// TIA Portal V20 export
// export: Created 2025-12-01T14:57:41.0235932Z, ExportSetting None, DisplayName Totally Integrated Automation Portal, DisplayVersion V20 Update 3, DisplayName TIA Portal Openness, DisplayVersion V20 Update 3, DisplayName TIA Portal Version Control Interface, DisplayVersion V20 Update 3, DisplayName STEP 7 Professional, DisplayVersion V20 Update 3, DisplayName STEP 7 Safety, DisplayVersion V20 Update 2, DisplayName WinCC Basic/Comfort/Advanced, DisplayVersion V20 Update 3, DisplayName WinCC Professional, DisplayVersion V20 Update 3, DisplayName WinCC Unified, DisplayVersion V20 Update 3
FUNCTION_BLOCK "FB385_Operaciones_Paletizador_NDD"   // FB385, LAD
{ S7_Optimized_Access := 'FALSE' }
// stored: AutoNumber false, SetENOAutomatically false
   VAR_INPUT
      MesaElevador : UInt;
      MesaGarra : UInt;
      MesaHorquilla : UInt;
      ZonaCajon_Libre : Bool;
      ElevadorEnReposo : Bool;
      ElevadorPaletizando : Bool;
      DesHabilitar_Horquilla : Bool;
      DesHabilitar_Garra : Bool;
   END_VAR
   VAR_IN_OUT
      Horquilla : "NDD_Interlock_Horquilla";
      Garra : "NDD_Interlock_Garras";
      TELEV : "NDD_Interlock_TElev";
      Ordenes : "NDD_Ordenes";
   END_VAR
   VAR
      ControlUT_MesaElevador : "UDT_UTs_Control";
      DatosUT_MesaElevador { S7_SetPoint := 'True'} : "UDT_UTs_Datos";
      ControlUT_MesaGarra { S7_SetPoint := 'True'} : "UDT_UTs_Control";
      ControlUT_MesaHorquilla { S7_SetPoint := 'True'} : "UDT_UTs_Control";
      UT_MesaElevador : UInt;
      UT_MesaGarra : UInt;
      UT_MesaHorquilla : UInt;
      DesHabilitar_NDD : Bool;
      ExisteUT_MTElev { ExternalAccessible := 'False'; ExternalVisible := 'False'; ExternalWritable := 'False'} : Bool;
      TElev_PaletizarPaleta : Bool;
      TElev_EvacuarPaleta : Bool;
      TElev_DestinoHorquilla : Bool;
      TElev_DestinoGarra : Bool;
      ExisteUT_MHorq { ExternalAccessible := 'False'; ExternalVisible := 'False'; ExternalWritable := 'False'} : Bool;
      Horq_DestinoGarra : Bool;
      ExisteUT_MGarra { ExternalAccessible := 'False'; ExternalVisible := 'False'; ExternalWritable := 'False'} : Bool;
      PeticionROBO_MGarra : Bool;
      Garra_DestinoElevador : Bool;
   END_VAR
   VAR_TEMP
      Guardar_AR1 : DWord;
      P_Temporal : DWord;
      Destino_MesaElevador : UInt;
      Destino_MesaHorquilla : UInt;
      Destino_MesaGarra : UInt;
      Numero_UT : UInt;
      ReturnValor : Int;
      Cero : Byte;
      EnCursoOperaciones : Bool;
   END_VAR
BEGIN

REGION Network 1: Inicializaciones
END_REGION

REGION Network 2: Contorl de DesHabilitar
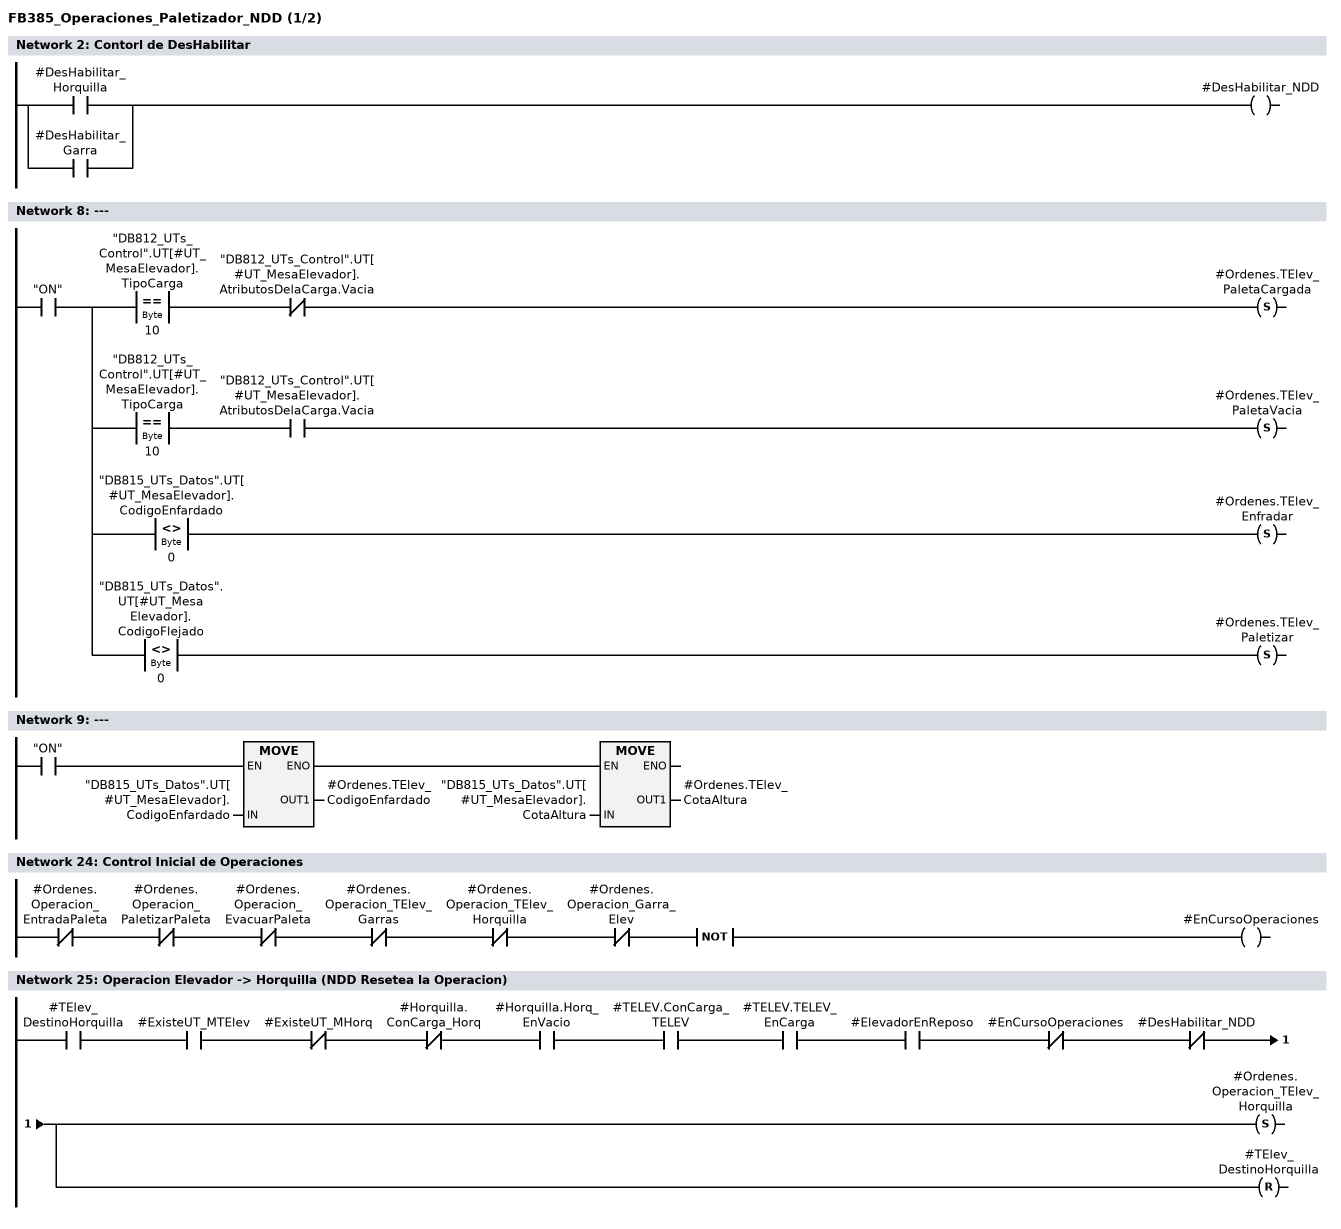
   RUNG wire#powerrail
      Contact( #DesHabilitar_Horquilla )
      wire#w1
      Coil( #DesHabilitar_NDD )
   END_RUNG
   RUNG wire#powerrail
      Contact( #DesHabilitar_Garra )
   END_RUNG wire#w1
   // the same network as SCL:
   #DesHabilitar_NDD := #DesHabilitar_Horquilla OR #DesHabilitar_Garra;
END_REGION

NETWORK
TITLE = Inicializar Variables Generales
/////////////////////////////////////////////////////////////////////////////
/////////////////////////////////////////////////////////////////////////////
// - Inicializaciones Generales
      L     #MesaElevador;  // Destino = Mesa del Elevador
      L     "CTE_OffsetMesa";
      +I;
      T     #Destino_MesaElevador;

      L     #MesaHorquilla;  // Destino = Mesa de la Horquilla
      L     "CTE_OffsetMesa";
      +I;
      T     #Destino_MesaHorquilla;

      L     #MesaGarra;  // Destino = Mesa de la Garra
      L     "CTE_OffsetMesa";
      +I;
      T     #Destino_MesaGarra;



NETWORK
TITLE = Lectura de Datos de la UT de la Mesa del Elevador
/////////////////////////////////////////////////////////////////////////////
/////////////////////////////////////////////////////////////////////////////
// - Inicializaciones Previas
      TAR1  #Guardar_AR1;  // - Guardar el AR1


// - Inicializaciones Variables
      SET;
      R     #Ordenes.TElev_PaletaCargada;
      R     #Ordenes.TElev_PaletaVacia;
      R     #Ordenes.TElev_Enfradar;
      R     #Ordenes.TElev_Paletizar;

      SET;
      R     #ExisteUT_MTElev;
      S     #Ordenes.TElev_SinUT;

      L     0;
      T     #Ordenes.TElev_CodigoEnfardado;
      T     #Ordenes.TElev_CotaAltura;

// - Borrado de datos UT en la Mesa del Elevador
      L     0;
      T     #Cero;
      CALL  FILL
      ( BVAL    := #Cero,
        RET_VAL := #ReturnValor,
        BLK     := #ControlUT_MesaElevador
      );
      CALL  FILL
      ( BVAL    := #Cero,
        RET_VAL := #ReturnValor,
        BLK     := #DatosUT_MesaElevador
      );



NETWORK
TITLE = ---
//////////////////////////////////////////////////////////////////////////////
//////////////////////////////////////////////////////////////////////////////
// - Recoger Datos de la Mesa
      L     "DB810_ColasMesas".Colas[#MesaElevador].UT_PrimeraMesa;
      T     #Numero_UT;

      L     #Numero_UT;
      L     0;
      ==I;
      JC    FinDatosUT_MTElev;  // - No hay UT's ?


//////////////////////////////////////////////////////////////////////////////
//////////////////////////////////////////////////////////////////////////////
// - Hay UT en la Mesa
      SET;
      R     #Ordenes.TElev_SinUT;
      S     #ExisteUT_MTElev;

      L     #Numero_UT;
      T     #UT_MesaElevador;

      CALL  BLKMOV
      ( SRCBLK  := "DB812_UTs_Control".UT[#UT_MesaElevador],
        RET_VAL := #ReturnValor,
        DSTBLK  := #ControlUT_MesaElevador
      );
      CALL  BLKMOV
      ( SRCBLK  := "DB815_UTs_Datos".UT[#UT_MesaElevador],
        RET_VAL := #ReturnValor,
        DSTBLK  := #DatosUT_MesaElevador
      );



NETWORK
TITLE = ---
/////////////////////////////////////////////////////////////////////////////
/////////////////////////////////////////////////////////////////////////////
// - Final de la Recogida de Datos
FinDatosUT_MTElev:NOP   0;
      LAR1  #Guardar_AR1;  // - Recuperar AR1



NETWORK
TITLE = Control de datos de la UT de la Mesa Elevadora
/////////////////////////////////////////////////////////////////////////////
/////////////////////////////////////////////////////////////////////////////
// - Si No Existe UT no hacer nada más
      SET;
      A     #ExisteUT_MTElev;
      JC    InicioControlDatosUT_MTElev;

      SET;
      R     #TElev_PaletizarPaleta;
      R     #TElev_EvacuarPaleta;
      R     #TElev_DestinoHorquilla;
      R     #TElev_DestinoGarra;

      JC    FinalControlDatosUT_MTElev;

// - Existe UT en la Mesa
InicioControlDatosUT_MTElev:NOP   0;



REGION Network 8: ---
   RUNG wire#powerrail
      Contact( "ON" )
      wire#w1
      { S7_Templates := "SrcType := Byte" } EQ_Contact(in1 := "DB812_UTs_Control".UT[#UT_MesaElevador].TipoCarga, in2 := 10)
      I_Contact( "DB812_UTs_Control".UT[#UT_MesaElevador].AtributosDelaCarga.Vacia )
      S_Coil( #Ordenes.TElev_PaletaCargada )
   END_RUNG
   RUNG wire#w1
      { S7_Templates := "SrcType := Byte" } EQ_Contact(in1 := "DB812_UTs_Control".UT[#UT_MesaElevador].TipoCarga, in2 := 10)
      Contact( "DB812_UTs_Control".UT[#UT_MesaElevador].AtributosDelaCarga.Vacia )
      S_Coil( #Ordenes.TElev_PaletaVacia )
   END_RUNG
   RUNG wire#w1
      { S7_Templates := "SrcType := Byte" } NE_Contact(in1 := "DB815_UTs_Datos".UT[#UT_MesaElevador].CodigoEnfardado, in2 := 0)
      S_Coil( #Ordenes.TElev_Enfradar )
   END_RUNG
   RUNG wire#w1
      { S7_Templates := "SrcType := Byte" } NE_Contact(in1 := "DB815_UTs_Datos".UT[#UT_MesaElevador].CodigoFlejado, in2 := 0)
      S_Coil( #Ordenes.TElev_Paletizar )
   END_RUNG
   // the same network as SCL:
   IF "ON" AND ("DB812_UTs_Control".UT[#UT_MesaElevador].TipoCarga = 10) AND NOT "DB812_UTs_Control".UT[#UT_MesaElevador].AtributosDelaCarga.Vacia THEN
       #Ordenes.TElev_PaletaCargada := TRUE;
   END_IF;
   IF "ON" AND ("DB812_UTs_Control".UT[#UT_MesaElevador].TipoCarga = 10) AND "DB812_UTs_Control".UT[#UT_MesaElevador].AtributosDelaCarga.Vacia THEN
       #Ordenes.TElev_PaletaVacia := TRUE;
   END_IF;
   IF "ON" AND ("DB815_UTs_Datos".UT[#UT_MesaElevador].CodigoEnfardado <> 0) THEN
       #Ordenes.TElev_Enfradar := TRUE;
   END_IF;
   IF "ON" AND ("DB815_UTs_Datos".UT[#UT_MesaElevador].CodigoFlejado <> 0) THEN
       #Ordenes.TElev_Paletizar := TRUE;
   END_IF;
END_REGION

REGION Network 9: ---
   RUNG wire#powerrail
      Contact( "ON" )
      Move(in := "DB815_UTs_Datos".UT[#UT_MesaElevador].CodigoEnfardado, out1 => #Ordenes.TElev_CodigoEnfardado)
      Move(in := "DB815_UTs_Datos".UT[#UT_MesaElevador].CotaAltura, out1 => #Ordenes.TElev_CotaAltura)
   END_RUNG
   // the same network as SCL:
   IF "ON" THEN
       #Ordenes.TElev_CodigoEnfardado := "DB815_UTs_Datos".UT[#UT_MesaElevador].CodigoEnfardado;
       #Ordenes.TElev_CotaAltura := "DB815_UTs_Datos".UT[#UT_MesaElevador].CotaAltura;
   END_IF;
END_REGION

NETWORK
TITLE = ---
//////////////////////////////////////////////////////////////////////////
//////////////////////////////////////////////////////////////////////////
// - Hay que general Orden en la Mesa
      SET;
      L     11;  // Ha cambiado de Mesa
      L     "DB812_UTs_Control".UT[#UT_MesaElevador].EstadoRecepcionUT;
      ==I;
      JC    InicioControlDestinoUT_MTElev;

      SET;
      L     13;  // Realizado Reset desde Panatalla
      L     "DB812_UTs_Control".UT[#UT_MesaElevador].EstadoRecepcionUT;
      ==I;
      JC    InicioControlDestinoUT_MTElev;

      SET;
      L     17;  // Ha Recibido Nueva Ruta
      L     "DB812_UTs_Control".UT[#UT_MesaElevador].EstadoRecepcionUT;
      ==I;
      JC    InicioControlDestinoUT_MTElev;


// - Activar el paletizado de la paleta
      SET;
      A     #Ordenes.TElev_Paletizar;
      S     #TElev_PaletizarPaleta;

      SET;
      AN    #Ordenes.TElev_Paletizar;
      R     #TElev_PaletizarPaleta;

// - No hay que generar orden
      JU    FinalControlDestinoUT_MTElev;


//////////////////////////////////////////////////////////////////////////
//////////////////////////////////////////////////////////////////////////
// - Inicio del Control del Destino
InicioControlDestinoUT_MTElev:NOP   0;

      SET;  // - Tiene Algun Destino Recibido
      L     "DB812_UTs_Control".UT[#UT_MesaElevador].MesaDestino;
      L     0;
      ==I;
      JC    FinalControlDestinoUT_MTElev;

      SET;  // - Tiene Destino la Mesa del Elevador
      L     "DB812_UTs_Control".UT[#UT_MesaElevador].MesaDestino;
      L     #Destino_MesaElevador;
      ==I;
      JC    DestinoUT_MesaElevadora_MTElev;

      SET;  // - Tiene Destino la Mesa de la Horquilla
      L     "DB812_UTs_Control".UT[#UT_MesaElevador].MesaDestino;
      L     #Destino_MesaHorquilla;
      ==I;
      JC    DestinoUT_MesaHorquilla_MTElev;

      SET;  // - Tiene Destino la Mesa de la Garra
      L     "DB812_UTs_Control".UT[#UT_MesaElevador].MesaDestino;
      L     #Destino_MesaGarra;
      ==I;
      JC    DestinoUT_MesaGarra_MTElev;

// - Tiene Destino fuera del NDD
      JU    DestinoUT_MesaSalida_MTElev;


//////////////////////////////////////////////////////////////////////////
//////////////////////////////////////////////////////////////////////////
// - Destino Mesa del Elevador
// ---- Pedir Ruta (21)
// ---- Activar Paletiza Paleta en el Elevador
DestinoUT_MesaElevadora_MTElev:NOP   0;
      L     "DB812_UTs_Control".UT[#UT_MesaElevador].EstadoGeneralUT;
      L     0;
      <>I;
      JC    FinalControlDestinoUT_MTElev;

      L     0;
      T     "DB812_UTs_Control".UT[#UT_MesaElevador].EstadoRecepcionUT;
      L     21;
      T     "DB812_UTs_Control".UT[#UT_MesaElevador].EstadoGeneralUT;

      JU    FinalControlDestinoUT_MTElev;


//////////////////////////////////////////////////////////////////////////
//////////////////////////////////////////////////////////////////////////
// - Destino Mesa de la Horquilla
// ---- Paleta con Destino la Horquilla
DestinoUT_MesaHorquilla_MTElev:NOP   0;
      L     0;
      T     "DB812_UTs_Control".UT[#UT_MesaElevador].EstadoRecepcionUT;

      SET;
      S     #TElev_DestinoHorquilla;

      JU    FinalControlDestinoUT_MTElev;


//////////////////////////////////////////////////////////////////////////
//////////////////////////////////////////////////////////////////////////
// - Destino Mesa de la Garra
// ---- Activar Paleta con Destino la Garra
DestinoUT_MesaGarra_MTElev:NOP   0;
      L     0;
      T     "DB812_UTs_Control".UT[#UT_MesaElevador].EstadoRecepcionUT;

      SET;
      S     #TElev_DestinoGarra;

      JU    FinalControlDestinoUT_MTElev;


//////////////////////////////////////////////////////////////////////////
//////////////////////////////////////////////////////////////////////////
// - Destino Mesa de Salida
// ---- Activar Evacuacion de la Paleta
DestinoUT_MesaSalida_MTElev:NOP   0;
      L     0;
      T     "DB812_UTs_Control".UT[#UT_MesaElevador].EstadoRecepcionUT;

      SET;
      S     #TElev_EvacuarPaleta;

      JU    FinalControlDestinoUT_MTElev;


//////////////////////////////////////////////////////////////////////////
//////////////////////////////////////////////////////////////////////////
// - Final del Control del Destino
FinalControlDestinoUT_MTElev:NOP   0;



NETWORK
TITLE = ---
/////////////////////////////////////////////////////////////////////////////
/////////////////////////////////////////////////////////////////////////////
// - Final del Control de datos de la UT de la Mesa Elevadora
FinalControlDatosUT_MTElev:NOP   0;



NETWORK
TITLE = Lectura de Datos de la UT de la Mesa de la Horquilla
/////////////////////////////////////////////////////////////////////////////
/////////////////////////////////////////////////////////////////////////////
// - Inicializaciones Previas
      TAR1  #Guardar_AR1;  // - Guardar el AR1


// - Inicializaciones Variables
      SET;
      R     #ExisteUT_MHorq;

// Borrado de UT en la Mesa de la Horquilla
      L     0;
      T     #Cero;
      CALL  FILL
      ( BVAL    := #Cero,
        RET_VAL := #ReturnValor,
        BLK     := #ControlUT_MesaHorquilla
      );



NETWORK
TITLE = ---
//////////////////////////////////////////////////////////////////////////////
//////////////////////////////////////////////////////////////////////////////
// - Recoger Datos de la Mesa
      L     "DB810_ColasMesas".Colas[#MesaHorquilla].UT_PrimeraMesa;
      T     #Numero_UT;

      L     #Numero_UT;
      L     0;
      ==I;
      JC    FinDatosUT_MHorquilla;  // - No hay UT's ?


//////////////////////////////////////////////////////////////////////////////
//////////////////////////////////////////////////////////////////////////////
// - Hay UT en la Mesa
      SET;
      S     #ExisteUT_MHorq;

      L     #Numero_UT;
      T     #UT_MesaHorquilla;
      CALL  BLKMOV
      ( SRCBLK  := "DB812_UTs_Control".UT[#UT_MesaHorquilla],
        RET_VAL := #ReturnValor,
        DSTBLK  := #ControlUT_MesaHorquilla
      );



NETWORK
TITLE = ---
/////////////////////////////////////////////////////////////////////////////
/////////////////////////////////////////////////////////////////////////////
// - Final de la Recogida de Datos

FinDatosUT_MHorquilla:NOP   0;
      LAR1  #Guardar_AR1;  // - Recuperar AR1




NETWORK
TITLE = Control de datos de la UT de la Mesa de Horquilla
/////////////////////////////////////////////////////////////////////////////
/////////////////////////////////////////////////////////////////////////////
// - Si No Existe UT no hacer nada más
      SET;
      A     #ExisteUT_MHorq;
      JC    InicioControlDatosUT_MHorquilla;

      SET;
      R     #Horq_DestinoGarra;

      JU    FinalControlDatosUT_MHorquilla;

// - Existe UT en la Mesa
InicioControlDatosUT_MHorquilla:NOP   0;



NETWORK
TITLE = ---
//////////////////////////////////////////////////////////////////////////
//////////////////////////////////////////////////////////////////////////
// - Hay que general Orden en la Mesa
      SET;
      L     11;  // Ha cambiado de Mesa
      L     "DB812_UTs_Control".UT[#UT_MesaHorquilla].EstadoEventoRecibido;
      ==I;
      JC    InicioControlDestinoUT_MHorquilla;

      SET;
      L     13;  // Realizado Reset desde Panatalla
      L     "DB812_UTs_Control".UT[#UT_MesaHorquilla].EstadoRecepcionUT;
      ==I;
      JC    InicioControlDestinoUT_MHorquilla;

      SET;
      L     17;  // Ha Recibido Nueva Ruta
      L     "DB812_UTs_Control".UT[#UT_MesaHorquilla].EstadoRecepcionUT;
      ==I;
      JC    InicioControlDestinoUT_MHorquilla;

// - No hay que generar orden
      JU    FinalControlDestinoUT_MHorquilla;


//////////////////////////////////////////////////////////////////////////
//////////////////////////////////////////////////////////////////////////
// - Inicio del Control del Destino
InicioControlDestinoUT_MHorquilla:NOP   0;

      SET;  // - Tiene Algun Destino Recibido
      L     "DB812_UTs_Control".UT[#UT_MesaHorquilla].MesaDestino;
      L     0;
      ==I;
      JC    FinalControlDestinoUT_MHorquilla;

      SET;  // - Tiene Destino la Mesa de la Horquilla
      L     "DB812_UTs_Control".UT[#UT_MesaHorquilla].MesaDestino;
      L     #Destino_MesaHorquilla;
      ==I;
      JC    DestinoUT_MesaHorquilla_MHorquilla;

      SET;  // - Tiene Destino la Mesa de la Garra
      L     "DB812_UTs_Control".UT[#UT_MesaHorquilla].MesaDestino;
      L     #Destino_MesaGarra;
      ==I;
      JC    DestinoUT_MesaGarra_MHorquilla;

// - No tiene destino de salida Previsto
      JU    FinalControlDestinoUT_MHorquilla;


//////////////////////////////////////////////////////////////////////////
//////////////////////////////////////////////////////////////////////////
// - Destino Mesa de la Horquilla
// ---- Pedir Ruta (21)
DestinoUT_MesaHorquilla_MHorquilla:NOP   0;
      SET;
      L     "DB812_UTs_Control".UT[#UT_MesaHorquilla].EstadoGeneralUT;
      L     0;
      <>I;
      JC    FinalControlDestinoUT_MHorquilla;

      L     0;
      T     "DB812_UTs_Control".UT[#UT_MesaHorquilla].EstadoRecepcionUT;
      L     21;
      T     "DB812_UTs_Control".UT[#UT_MesaHorquilla].EstadoGeneralUT;

      JU    FinalControlDestinoUT_MHorquilla;


//////////////////////////////////////////////////////////////////////////
//////////////////////////////////////////////////////////////////////////
// - Destino Mesa de la Garra
// ---- Activar Paleta con Destino la Garra
DestinoUT_MesaGarra_MHorquilla:NOP   0;
      L     0;
      T     "DB812_UTs_Control".UT[#UT_MesaHorquilla].EstadoRecepcionUT;

      SET;
      S     #Horq_DestinoGarra;

      JU    FinalControlDestinoUT_MHorquilla;


//////////////////////////////////////////////////////////////////////////
//////////////////////////////////////////////////////////////////////////
// - Final del Control del Destino
FinalControlDestinoUT_MHorquilla:NOP   0;



NETWORK
TITLE = ---
/////////////////////////////////////////////////////////////////////////////
/////////////////////////////////////////////////////////////////////////////
// - Final del Control de datos de la UT de la Mesa de la Horquilla
FinalControlDatosUT_MHorquilla:NOP   0;



NETWORK
TITLE = Lectura de Datos de la UT de la Mesa de la Garra
/////////////////////////////////////////////////////////////////////////////
/////////////////////////////////////////////////////////////////////////////
// - Inicializaciones Previas
      TAR1  #Guardar_AR1;  // - Guardar el AR1


// - Inicializaciones Variables
      SET;
      R     #ExisteUT_MGarra;

// - Borrado de Datos UT en la Mesa de la Garra
      L     0;
      T     #Cero;
      CALL  FILL
      ( BVAL    := #Cero,
        RET_VAL := #ReturnValor,
        BLK     := #ControlUT_MesaGarra
      );



NETWORK
TITLE = ---
//////////////////////////////////////////////////////////////////////////////
//////////////////////////////////////////////////////////////////////////////
// - Recoger Datos de la Mesa
      L     "DB810_ColasMesas".Colas[#MesaGarra].UT_PrimeraMesa;
      T     #Numero_UT;

      L     #Numero_UT;
      L     0;
      ==I;
      JC    FinDatosUT_MGarra;  // - No hay UT's ?


//////////////////////////////////////////////////////////////////////////////
//////////////////////////////////////////////////////////////////////////////
// - Hay UT en la Mesa
      SET;
      S     #ExisteUT_MGarra;

      L     #Numero_UT;
      T     #UT_MesaGarra;

      CALL  BLKMOV
      ( SRCBLK  := "DB812_UTs_Control".UT[#UT_MesaGarra],
        RET_VAL := #ReturnValor,
        DSTBLK  := #ControlUT_MesaGarra
      );



NETWORK
TITLE = ---
/////////////////////////////////////////////////////////////////////////////
/////////////////////////////////////////////////////////////////////////////
// - Final de la Recogida de Datos
FinDatosUT_MGarra:NOP   0;
      LAR1  #Guardar_AR1;  // - Recuperar AR1



NETWORK
TITLE = Control de datos de la UT de la Mesa de Garra
/////////////////////////////////////////////////////////////////////////////
/////////////////////////////////////////////////////////////////////////////
// - Si No Existe UT no hacer nada más
      SET;
      A     #ExisteUT_MGarra;
      JC    InicioControlDatosUT_MGarra;

      SET;
      R     #Garra_DestinoElevador;
      R     #PeticionROBO_MGarra;

      JU    FinalControlDatosUT_MGarra;

// - Existe UT en la Mesa
InicioControlDatosUT_MGarra:NOP   0;



NETWORK
TITLE = ---
//////////////////////////////////////////////////////////////////////////
//////////////////////////////////////////////////////////////////////////
// - Hay que general Orden en la Mesa
      SET;
      L     11;  // Ha cambiado de Mesa
      L     "DB812_UTs_Control".UT[#UT_MesaGarra].EstadoRecepcionUT;
      ==I;
      JC    InicioControlDestinoUT_MGarra;

      SET;
      L     13;  // Realizado Reset desde Panatalla
      L     "DB812_UTs_Control".UT[#UT_MesaGarra].EstadoRecepcionUT;
      ==I;
      JC    InicioControlDestinoUT_MGarra;

      SET;
      L     17;  // Ha Recibido Nueva Ruta
      L     "DB812_UTs_Control".UT[#UT_MesaGarra].EstadoRecepcionUT;
      ==I;
      JC    InicioControlDestinoUT_MGarra;

// - Ha llegado al final de Paletizado en la Garra
      SET;
      A     #Garra.PosGarrasTransfer_OK;
      AN    #PeticionROBO_MGarra;
      JC    FinPaletizadoEnGarra;


// - No hay que generar orden
      JU    FinalControlDestinoUT_MGarra;

//////////////////////////////////////////////////////////////////////////
//////////////////////////////////////////////////////////////////////////
// - Final de Paletizado En Garra
// - Peticicion de Ruta - Motivo ROBO
FinPaletizadoEnGarra:NOP   0;

// - Pedir la Evacuacion de la Mesa de la Garra en la UT
      L     "DB812_UTs_Control".UT[#UT_MesaGarra].MesaDestino;
      L     0;
      ==I;
      JC    PedirRuta_ControlDestinoUT_MGarra;

      L     "DB812_UTs_Control".UT[#UT_MesaGarra].MesaDestino;
      L     #Destino_MesaGarra;
      <>I;
      JC    FinalControlDestinoUT_MGarra;

PedirRuta_ControlDestinoUT_MGarra:NOP   0;
      L     "DB812_UTs_Control".UT[#UT_MesaGarra].EstadoEventoAGenerar;
      L     0;
      <>I;
      JC    FinalControlDestinoUT_MGarra;

      L     126;  // Peticion de Ruta - Motivo ROBO
      T     "DB812_UTs_Control".UT[#UT_MesaGarra].EstadoEventoAGenerar;

      SET;
      S     #PeticionROBO_MGarra;

      JU    FinalControlDestinoUT_MGarra;

//////////////////////////////////////////////////////////////////////////
//////////////////////////////////////////////////////////////////////////
// - Inicio del Control del Destino
InicioControlDestinoUT_MGarra:NOP   0;
      SET;  // - Tiene Algun Destino Recibido
      L     "DB812_UTs_Control".UT[#UT_MesaGarra].MesaDestino;
      L     0;
      ==I;
      JC    FinalControlDestinoUT_MGarra;

// - Tiene Destino la Mesa de la Garra
      L     "DB812_UTs_Control".UT[#UT_MesaGarra].MesaDestino;
      L     #Destino_MesaGarra;
      ==I;
      JC    DestinoUT_MesaGarra_MGarra;


// - Tiene Destino de Evacuacion de la Mesa de la Garra
      JU    DestinoUT_MesaSalida_MGarra;


//////////////////////////////////////////////////////////////////////////
//////////////////////////////////////////////////////////////////////////
// - Destino Mesa de la Garra
// ---- Pedir Ruta (21)
DestinoUT_MesaGarra_MGarra:NOP   0;
      SET;
      L     "DB812_UTs_Control".UT[#UT_MesaGarra].EstadoGeneralUT;
      L     0;
      <>I;
      JC    FinalControlDestinoUT_MGarra;

      L     0;
      T     "DB812_UTs_Control".UT[#UT_MesaGarra].EstadoRecepcionUT;
      L     21;
      T     "DB812_UTs_Control".UT[#UT_MesaGarra].EstadoGeneralUT;

      SET;
      R     #PeticionROBO_MGarra;

      JU    FinalControlDestinoUT_MGarra;


//////////////////////////////////////////////////////////////////////////
//////////////////////////////////////////////////////////////////////////
// - Destino Fuera de la Mesa de la Garra
// ---- Activar Paleta con Destino el Elevador
DestinoUT_MesaSalida_MGarra:NOP   0;
      L     0;
      T     "DB812_UTs_Control".UT[#UT_MesaGarra].EstadoRecepcionUT;

      SET;
      S     #Garra_DestinoElevador;
      R     #PeticionROBO_MGarra;

      JU    FinalControlDestinoUT_MGarra;


//////////////////////////////////////////////////////////////////////////
//////////////////////////////////////////////////////////////////////////
// - Final del Control del Destino
FinalControlDestinoUT_MGarra:NOP   0;



NETWORK
TITLE = ---
/////////////////////////////////////////////////////////////////////////////
/////////////////////////////////////////////////////////////////////////////
// - Final del Control de datos de la UT de la Mesa de la Garra

FinalControlDatosUT_MGarra:NOP   0;



REGION Network 24: Control Inicial de Operaciones
   RUNG wire#powerrail
      I_Contact( #Ordenes.Operacion_EntradaPaleta )
      I_Contact( #Ordenes.Operacion_PaletizarPaleta )
      I_Contact( #Ordenes.Operacion_EvacuarPaleta )
      I_Contact( #Ordenes.Operacion_TElev_Garras )
      I_Contact( #Ordenes.Operacion_TElev_Horquilla )
      I_Contact( #Ordenes.Operacion_Garra_Elev )
      Not()
      Coil( #EnCursoOperaciones )
   END_RUNG
   // the same network as SCL:
   #EnCursoOperaciones := NOT (NOT #Ordenes.Operacion_EntradaPaleta AND NOT #Ordenes.Operacion_PaletizarPaleta AND NOT #Ordenes.Operacion_EvacuarPaleta AND NOT #Ordenes.Operacion_TElev_Garras AND NOT #Ordenes.Operacion_TElev_Horquilla AND NOT #Ordenes.Operacion_Garra_Elev);
END_REGION

REGION Network 25: Operacion Elevador -> Horquilla (NDD Resetea la Operacion)
   RUNG wire#powerrail
      Contact( #TElev_DestinoHorquilla )
      Contact( #ExisteUT_MTElev )
      I_Contact( #ExisteUT_MHorq )
      I_Contact( #Horquilla.ConCarga_Horq )
      Contact( #Horquilla.Horq_EnVacio )
      Contact( #TELEV.ConCarga_TELEV )
      Contact( #TELEV.TELEV_EnCarga )
      Contact( #ElevadorEnReposo )
      I_Contact( #EnCursoOperaciones )
      I_Contact( #DesHabilitar_NDD )
      wire#w1
      S_Coil( #Ordenes.Operacion_TElev_Horquilla )
   END_RUNG
   RUNG wire#w1
      R_Coil( #TElev_DestinoHorquilla )
   END_RUNG
   // the same network as SCL:
   IF #TElev_DestinoHorquilla AND #ExisteUT_MTElev AND NOT #ExisteUT_MHorq AND NOT #Horquilla.ConCarga_Horq AND #Horquilla.Horq_EnVacio AND #TELEV.ConCarga_TELEV AND #TELEV.TELEV_EnCarga AND #ElevadorEnReposo AND NOT #EnCursoOperaciones AND NOT #DesHabilitar_NDD THEN
       #Ordenes.Operacion_TElev_Horquilla := TRUE;
       #TElev_DestinoHorquilla := FALSE;
   END_IF;
END_REGION

REGION Network 26: Operacion Elevador -> Garra (NDD Resetea la Operacion)
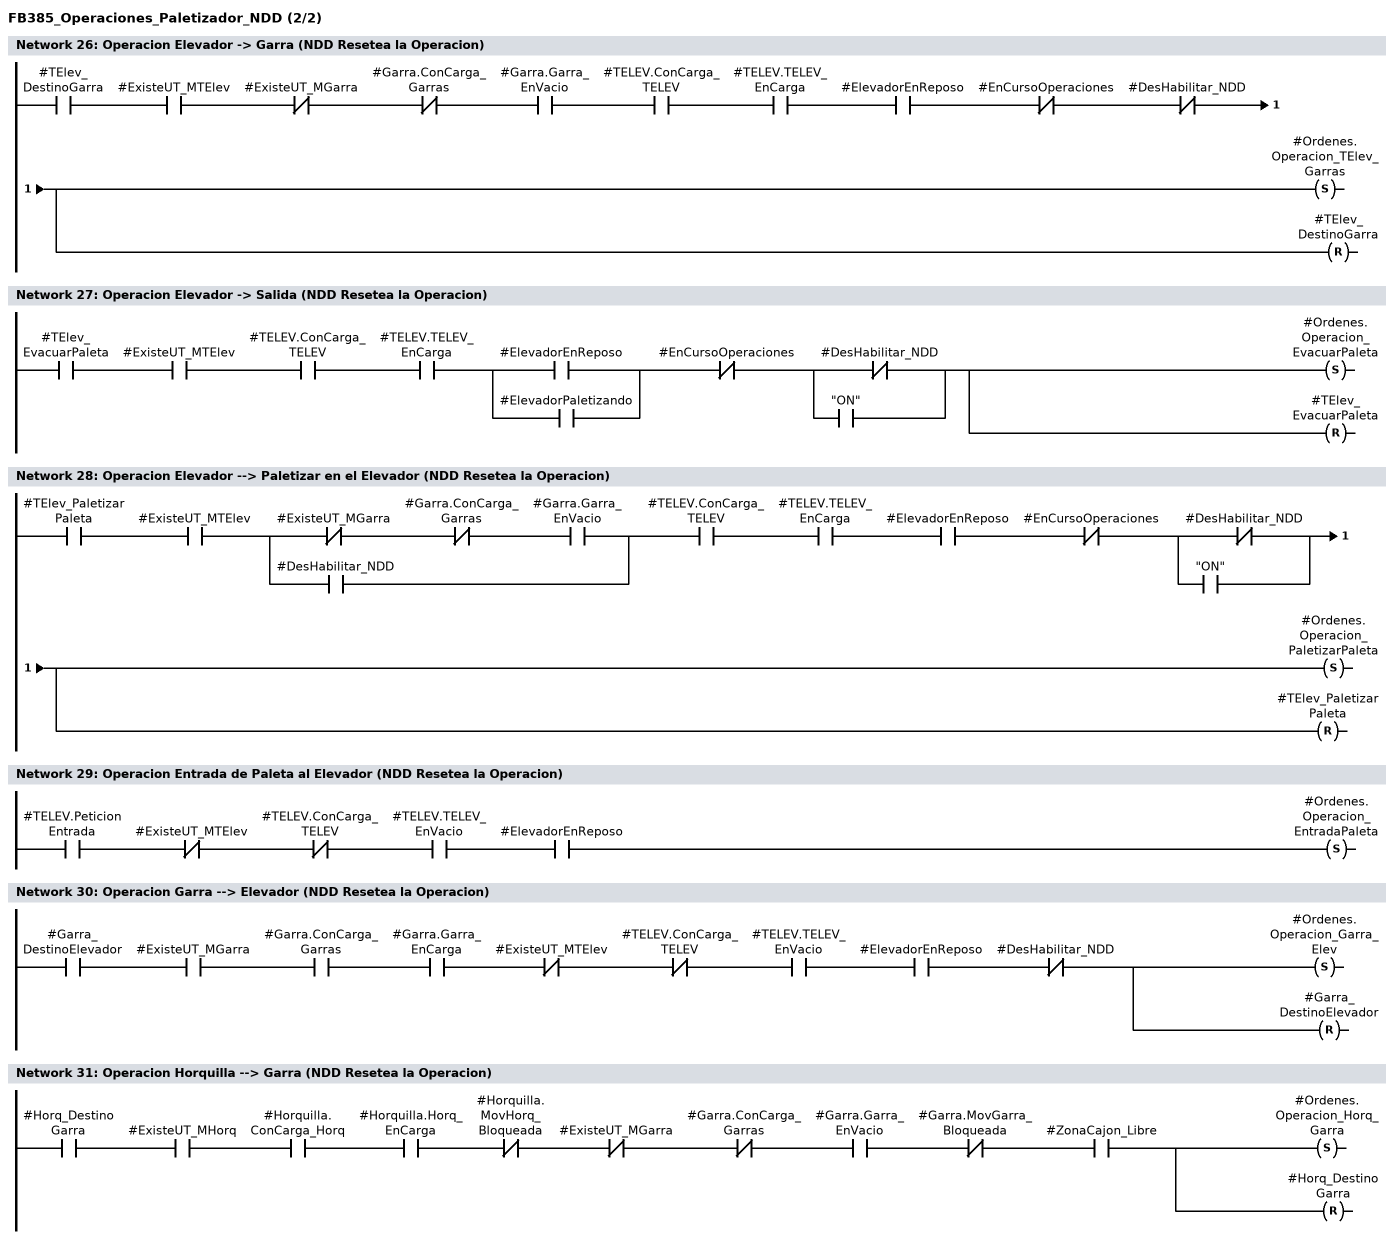
   RUNG wire#powerrail
      Contact( #TElev_DestinoGarra )
      Contact( #ExisteUT_MTElev )
      I_Contact( #ExisteUT_MGarra )
      I_Contact( #Garra.ConCarga_Garras )
      Contact( #Garra.Garra_EnVacio )
      Contact( #TELEV.ConCarga_TELEV )
      Contact( #TELEV.TELEV_EnCarga )
      Contact( #ElevadorEnReposo )
      I_Contact( #EnCursoOperaciones )
      I_Contact( #DesHabilitar_NDD )
      wire#w1
      S_Coil( #Ordenes.Operacion_TElev_Garras )
   END_RUNG
   RUNG wire#w1
      R_Coil( #TElev_DestinoGarra )
   END_RUNG
   // the same network as SCL:
   IF #TElev_DestinoGarra AND #ExisteUT_MTElev AND NOT #ExisteUT_MGarra AND NOT #Garra.ConCarga_Garras AND #Garra.Garra_EnVacio AND #TELEV.ConCarga_TELEV AND #TELEV.TELEV_EnCarga AND #ElevadorEnReposo AND NOT #EnCursoOperaciones AND NOT #DesHabilitar_NDD THEN
       #Ordenes.Operacion_TElev_Garras := TRUE;
       #TElev_DestinoGarra := FALSE;
   END_IF;
END_REGION

REGION Network 27: Operacion Elevador -> Salida (NDD Resetea la Operacion)
   RUNG wire#powerrail
      Contact( #TElev_EvacuarPaleta )
      Contact( #ExisteUT_MTElev )
      Contact( #TELEV.ConCarga_TELEV )
      Contact( #TELEV.TELEV_EnCarga )
      wire#w1
      Contact( #ElevadorEnReposo )
      wire#w2
      I_Contact( #EnCursoOperaciones )
      wire#w3
      I_Contact( #DesHabilitar_NDD )
      wire#w4
      S_Coil( #Ordenes.Operacion_EvacuarPaleta )
   END_RUNG
   RUNG wire#w1
      Contact( #ElevadorPaletizando )
   END_RUNG wire#w2
   RUNG wire#w3
      Contact( "ON" )
   END_RUNG wire#w4
   RUNG wire#w4
      R_Coil( #TElev_EvacuarPaleta )
   END_RUNG
   // the same network as SCL:
   IF #TElev_EvacuarPaleta AND #ExisteUT_MTElev AND #TELEV.ConCarga_TELEV AND #TELEV.TELEV_EnCarga AND (#ElevadorEnReposo OR #ElevadorPaletizando) AND NOT #EnCursoOperaciones AND (NOT #DesHabilitar_NDD OR "ON") THEN
       #Ordenes.Operacion_EvacuarPaleta := TRUE;
       #TElev_EvacuarPaleta := FALSE;
   END_IF;
END_REGION

REGION Network 28: Operacion Elevador --> Paletizar en el Elevador (NDD Resetea la Operacion)
   RUNG wire#powerrail
      Contact( #TElev_PaletizarPaleta )
      Contact( #ExisteUT_MTElev )
      wire#w1
      I_Contact( #ExisteUT_MGarra )
      I_Contact( #Garra.ConCarga_Garras )
      Contact( #Garra.Garra_EnVacio )
      wire#w2
      Contact( #TELEV.ConCarga_TELEV )
      Contact( #TELEV.TELEV_EnCarga )
      Contact( #ElevadorEnReposo )
      I_Contact( #EnCursoOperaciones )
      wire#w3
      I_Contact( #DesHabilitar_NDD )
      wire#w4
      S_Coil( #Ordenes.Operacion_PaletizarPaleta )
   END_RUNG
   RUNG wire#w1
      Contact( #DesHabilitar_NDD )
   END_RUNG wire#w2
   RUNG wire#w3
      Contact( "ON" )
   END_RUNG wire#w4
   RUNG wire#w4
      R_Coil( #TElev_PaletizarPaleta )
   END_RUNG
   // the same network as SCL:
   IF #TElev_PaletizarPaleta AND #ExisteUT_MTElev AND ((NOT #ExisteUT_MGarra AND NOT #Garra.ConCarga_Garras AND #Garra.Garra_EnVacio) OR #DesHabilitar_NDD) AND #TELEV.ConCarga_TELEV AND #TELEV.TELEV_EnCarga AND #ElevadorEnReposo AND NOT #EnCursoOperaciones AND (NOT #DesHabilitar_NDD OR "ON") THEN
       #Ordenes.Operacion_PaletizarPaleta := TRUE;
       #TElev_PaletizarPaleta := FALSE;
   END_IF;
END_REGION

REGION Network 29: Operacion Entrada de Paleta al Elevador (NDD Resetea la Operacion)
   RUNG wire#powerrail
      Contact( #TELEV.PeticionEntrada )
      I_Contact( #ExisteUT_MTElev )
      I_Contact( #TELEV.ConCarga_TELEV )
      Contact( #TELEV.TELEV_EnVacio )
      Contact( #ElevadorEnReposo )
      S_Coil( #Ordenes.Operacion_EntradaPaleta )
   END_RUNG
   // the same network as SCL:
   IF #TELEV.PeticionEntrada AND NOT #ExisteUT_MTElev AND NOT #TELEV.ConCarga_TELEV AND #TELEV.TELEV_EnVacio AND #ElevadorEnReposo THEN
       #Ordenes.Operacion_EntradaPaleta := TRUE;
   END_IF;
END_REGION

REGION Network 30: Operacion Garra --> Elevador (NDD Resetea la Operacion)
   RUNG wire#powerrail
      Contact( #Garra_DestinoElevador )
      Contact( #ExisteUT_MGarra )
      Contact( #Garra.ConCarga_Garras )
      Contact( #Garra.Garra_EnCarga )
      I_Contact( #ExisteUT_MTElev )
      I_Contact( #TELEV.ConCarga_TELEV )
      Contact( #TELEV.TELEV_EnVacio )
      Contact( #ElevadorEnReposo )
      I_Contact( #DesHabilitar_NDD )
      wire#w1
      S_Coil( #Ordenes.Operacion_Garra_Elev )
   END_RUNG
   RUNG wire#w1
      R_Coil( #Garra_DestinoElevador )
   END_RUNG
   // the same network as SCL:
   IF #Garra_DestinoElevador AND #ExisteUT_MGarra AND #Garra.ConCarga_Garras AND #Garra.Garra_EnCarga AND NOT #ExisteUT_MTElev AND NOT #TELEV.ConCarga_TELEV AND #TELEV.TELEV_EnVacio AND #ElevadorEnReposo AND NOT #DesHabilitar_NDD THEN
       #Ordenes.Operacion_Garra_Elev := TRUE;
       #Garra_DestinoElevador := FALSE;
   END_IF;
END_REGION

REGION Network 31: Operacion Horquilla --> Garra (NDD Resetea la Operacion)
   RUNG wire#powerrail
      Contact( #Horq_DestinoGarra )
      Contact( #ExisteUT_MHorq )
      Contact( #Horquilla.ConCarga_Horq )
      Contact( #Horquilla.Horq_EnCarga )
      I_Contact( #Horquilla.MovHorq_Bloqueada )
      I_Contact( #ExisteUT_MGarra )
      I_Contact( #Garra.ConCarga_Garras )
      Contact( #Garra.Garra_EnVacio )
      I_Contact( #Garra.MovGarra_Bloqueada )
      Contact( #ZonaCajon_Libre )
      wire#w1
      S_Coil( #Ordenes.Operacion_Horq_Garra )
   END_RUNG
   RUNG wire#w1
      R_Coil( #Horq_DestinoGarra )
   END_RUNG
   // the same network as SCL:
   IF #Horq_DestinoGarra AND #ExisteUT_MHorq AND #Horquilla.ConCarga_Horq AND #Horquilla.Horq_EnCarga AND NOT #Horquilla.MovHorq_Bloqueada AND NOT #ExisteUT_MGarra AND NOT #Garra.ConCarga_Garras AND #Garra.Garra_EnVacio AND NOT #Garra.MovGarra_Bloqueada AND #ZonaCajon_Libre THEN
       #Ordenes.Operacion_Horq_Garra := TRUE;
       #Horq_DestinoGarra := FALSE;
   END_IF;
END_REGION
END_FUNCTION_BLOCK
